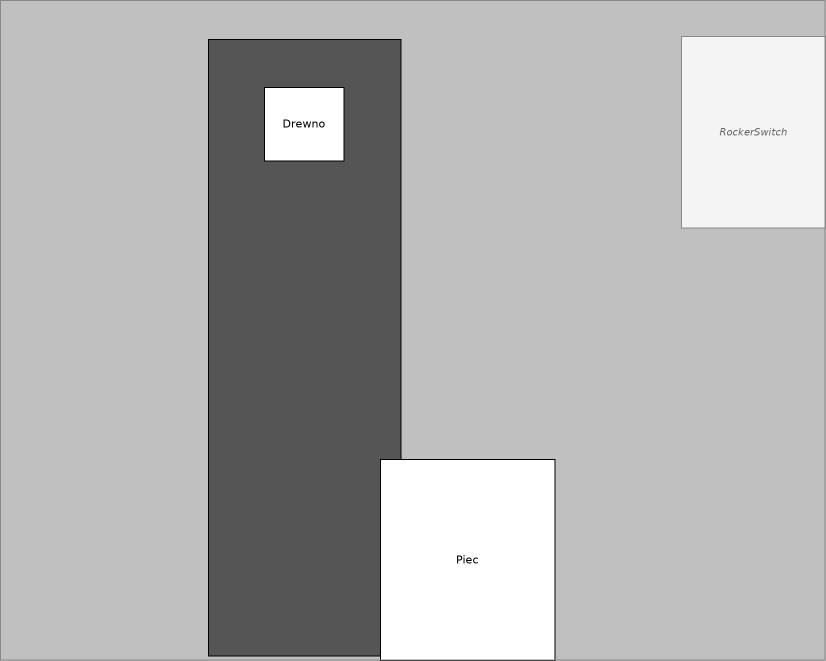
VISUALIZATION Ekran1  // 826x661
    Rectangle (208,39 193x617)
    Rectangle (264,87 80x74), "Drewno"
        p3560616238: MAIN.cola.pozycjaHoruzontalna
        p2738717112: MAIN.cola.pozycjaWzdluz
    RoundedRectangle (380,459 175x202), "Piec"
    RockerSwitch (681,36 145x192), variable: DVL.stanprzycisku, behaviour: TOGGLE, style: Switch-RockerSwitch-Gray
END_VISUALIZATION

(* stored: Version 1.1.0.1, ProductVersion 3.1.4024.4
   Visu Ekran1: Id {3a3464e0-66bc-4a1b-b790-9af29ffc465d} *)
